FUNCTION_BLOCK L5_prisavka_FBD
VAR_INPUT
	TL: BOOL;
	C1DPR: BOOL;
	CPC0: BOOL;
	CPC1:BOOL;
END_VAR
VAR_OUTPUT
	M1DPR: BOOL;
	RPC0: BOOL;
	RPC1: BOOL;
	RPS2: BOOL;
END_VAR
VAR
END_VAR

// NETWORK 1

END_FUNCTION_BLOCK

(* stored: Version 1.1.0.1, ProductVersion 3.1.4024.13
   POU L5_prisavka_FBD: Id {77402afc-242d-4fa8-b270-9c0e2d02378e}, SpecialFunc None *)
